BEGIN
   Info_Manag.P_Byte_First_Info := 20;
   Info_Manag.No_of_Infos := 30;
   Info_Manag.Len_Info := 24;
   Para_CMD[1].S_DB_No := 402;
   Para_CMD[1].S_Adress := 800;
   Para_CMD[1].D_Line := 1;
   Para_CMD[1].D_ASDU := 25860;
   Para_CMD[1].D_Info := 8;
   Para_CMD[1].Timeout := 10;
   Para_CMD[1].TI := 45;
   Para_CMD[1].Value := DWORD#16#0000_0005;
   Para_CMD[1].Termination_Type := 2;
   Para_CMD[2].S_DB_No := 402;
   Para_CMD[2].S_Adress := 816;
   Para_CMD[2].D_Line := 1;
   Para_CMD[2].D_ASDU := 25860;
   Para_CMD[2].D_Info := 9;
   Para_CMD[2].Timeout := 10;
   Para_CMD[2].TI := 45;
   Para_CMD[2].Value := DWORD#16#0000_0005;
   Para_CMD[2].Termination_Type := 2;
   Para_CMD[3].S_DB_No := 402;
   Para_CMD[3].S_Adress := 2016;
   Para_CMD[3].D_Line := 1;
   Para_CMD[3].D_ASDU := 26116;
   Para_CMD[3].D_Info := 8;
   Para_CMD[3].Timeout := 10;
   Para_CMD[3].TI := 45;
   Para_CMD[3].Value := DWORD#16#0000_0005;
   Para_CMD[3].Termination_Type := 2;
   Para_CMD[4].S_DB_No := 402;
   Para_CMD[4].S_Adress := 2032;
   Para_CMD[4].D_Line := 1;
   Para_CMD[4].D_ASDU := 26116;
   Para_CMD[4].D_Info := 9;
   Para_CMD[4].Timeout := 10;
   Para_CMD[4].TI := 45;
   Para_CMD[4].Value := DWORD#16#0000_0005;
   Para_CMD[4].Termination_Type := 2;
   Para_CMD[5].S_DB_No := 402;
   Para_CMD[5].S_Adress := 3232;
   Para_CMD[5].D_Line := 1;
   Para_CMD[5].D_ASDU := 26372;
   Para_CMD[5].D_Info := 8;
   Para_CMD[5].Timeout := 10;
   Para_CMD[5].TI := 45;
   Para_CMD[5].Value := DWORD#16#0000_0005;
   Para_CMD[5].Termination_Type := 2;
   Para_CMD[6].S_DB_No := 402;
   Para_CMD[6].S_Adress := 3248;
   Para_CMD[6].D_Line := 1;
   Para_CMD[6].D_ASDU := 26372;
   Para_CMD[6].D_Info := 9;
   Para_CMD[6].Timeout := 10;
   Para_CMD[6].TI := 45;
   Para_CMD[6].Value := DWORD#16#0000_0005;
   Para_CMD[6].Termination_Type := 2;
   Para_CMD[7].S_DB_No := 402;
   Para_CMD[7].S_Adress := 4448;
   Para_CMD[7].D_Line := 1;
   Para_CMD[7].D_ASDU := 26628;
   Para_CMD[7].D_Info := 8;
   Para_CMD[7].Timeout := 10;
   Para_CMD[7].TI := 45;
   Para_CMD[7].Value := DWORD#16#0000_0005;
   Para_CMD[7].Termination_Type := 2;
   Para_CMD[8].S_DB_No := 402;
   Para_CMD[8].S_Adress := 4464;
   Para_CMD[8].D_Line := 1;
   Para_CMD[8].D_ASDU := 26628;
   Para_CMD[8].D_Info := 9;
   Para_CMD[8].Timeout := 10;
   Para_CMD[8].TI := 45;
   Para_CMD[8].Value := DWORD#16#0000_0005;
   Para_CMD[8].Termination_Type := 2;
   Para_CMD[9].S_DB_No := 402;
   Para_CMD[9].S_Adress := 5664;
   Para_CMD[9].D_Line := 1;
   Para_CMD[9].D_ASDU := 26884;
   Para_CMD[9].D_Info := 8;
   Para_CMD[9].Timeout := 10;
   Para_CMD[9].TI := 45;
   Para_CMD[9].Value := DWORD#16#0000_0005;
   Para_CMD[9].Termination_Type := 2;
   Para_CMD[10].S_DB_No := 402;
   Para_CMD[10].S_Adress := 5680;
   Para_CMD[10].D_Line := 1;
   Para_CMD[10].D_ASDU := 26884;
   Para_CMD[10].D_Info := 9;
   Para_CMD[10].Timeout := 10;
   Para_CMD[10].TI := 45;
   Para_CMD[10].Value := DWORD#16#0000_0005;
   Para_CMD[10].Termination_Type := 2;
   Para_CMD[11].S_DB_No := 402;
   Para_CMD[11].S_Adress := 6880;
   Para_CMD[11].D_Line := 1;
   Para_CMD[11].D_ASDU := 27140;
   Para_CMD[11].D_Info := 8;
   Para_CMD[11].Timeout := 10;
   Para_CMD[11].TI := 45;
   Para_CMD[11].Value := DWORD#16#0000_0005;
   Para_CMD[11].Termination_Type := 2;
   Para_CMD[12].S_DB_No := 402;
   Para_CMD[12].S_Adress := 6896;
   Para_CMD[12].D_Line := 1;
   Para_CMD[12].D_ASDU := 27140;
   Para_CMD[12].D_Info := 9;
   Para_CMD[12].Timeout := 10;
   Para_CMD[12].TI := 45;
   Para_CMD[12].Value := DWORD#16#0000_0005;
   Para_CMD[12].Termination_Type := 2;
   Para_CMD[13].S_DB_No := 402;
   Para_CMD[13].S_Adress := 8096;
   Para_CMD[13].D_Line := 1;
   Para_CMD[13].D_ASDU := 27396;
   Para_CMD[13].D_Info := 8;
   Para_CMD[13].Timeout := 10;
   Para_CMD[13].TI := 45;
   Para_CMD[13].Value := DWORD#16#0000_0005;
   Para_CMD[13].Termination_Type := 2;
   Para_CMD[14].S_DB_No := 402;
   Para_CMD[14].S_Adress := 8112;
   Para_CMD[14].D_Line := 1;
   Para_CMD[14].D_ASDU := 27396;
   Para_CMD[14].D_Info := 9;
   Para_CMD[14].Timeout := 10;
   Para_CMD[14].TI := 45;
   Para_CMD[14].Value := DWORD#16#0000_0005;
   Para_CMD[14].Termination_Type := 2;
   Para_CMD[15].S_DB_No := 402;
   Para_CMD[15].S_Adress := 9312;
   Para_CMD[15].D_Line := 1;
   Para_CMD[15].D_ASDU := 27652;
   Para_CMD[15].D_Info := 8;
   Para_CMD[15].Timeout := 10;
   Para_CMD[15].TI := 45;
   Para_CMD[15].Value := DWORD#16#0000_0005;
   Para_CMD[15].Termination_Type := 2;
   Para_CMD[16].S_DB_No := 402;
   Para_CMD[16].S_Adress := 9328;
   Para_CMD[16].D_Line := 1;
   Para_CMD[16].D_ASDU := 27652;
   Para_CMD[16].D_Info := 9;
   Para_CMD[16].Timeout := 10;
   Para_CMD[16].TI := 45;
   Para_CMD[16].Value := DWORD#16#0000_0005;
   Para_CMD[16].Termination_Type := 2;
   Para_CMD[17].S_DB_No := 402;
   Para_CMD[17].S_Adress := 10528;
   Para_CMD[17].D_Line := 1;
   Para_CMD[17].D_ASDU := 28164;
   Para_CMD[17].D_Info := 8;
   Para_CMD[17].Timeout := 10;
   Para_CMD[17].TI := 45;
   Para_CMD[17].Value := DWORD#16#0000_0005;
   Para_CMD[17].Termination_Type := 2;
   Para_CMD[18].S_DB_No := 402;
   Para_CMD[18].S_Adress := 10544;
   Para_CMD[18].D_Line := 1;
   Para_CMD[18].D_ASDU := 28164;
   Para_CMD[18].D_Info := 9;
   Para_CMD[18].Timeout := 10;
   Para_CMD[18].TI := 45;
   Para_CMD[18].Value := DWORD#16#0000_0005;
   Para_CMD[18].Termination_Type := 2;
   Para_CMD[19].S_DB_No := 402;
   Para_CMD[19].S_Adress := 11744;
   Para_CMD[19].D_Line := 1;
   Para_CMD[19].D_ASDU := 28420;
   Para_CMD[19].D_Info := 8;
   Para_CMD[19].Timeout := 10;
   Para_CMD[19].TI := 45;
   Para_CMD[19].Value := DWORD#16#0000_0005;
   Para_CMD[19].Termination_Type := 2;
   Para_CMD[20].S_DB_No := 402;
   Para_CMD[20].S_Adress := 11760;
   Para_CMD[20].D_Line := 1;
   Para_CMD[20].D_ASDU := 28420;
   Para_CMD[20].D_Info := 9;
   Para_CMD[20].Timeout := 10;
   Para_CMD[20].TI := 45;
   Para_CMD[20].Value := DWORD#16#0000_0005;
   Para_CMD[20].Termination_Type := 2;
   Para_CMD[21].S_DB_No := 402;
   Para_CMD[21].S_Adress := 12960;
   Para_CMD[21].D_Line := 1;
   Para_CMD[21].D_ASDU := 28676;
   Para_CMD[21].D_Info := 8;
   Para_CMD[21].Timeout := 10;
   Para_CMD[21].TI := 45;
   Para_CMD[21].Value := DWORD#16#0000_0005;
   Para_CMD[21].Termination_Type := 2;
   Para_CMD[22].S_DB_No := 402;
   Para_CMD[22].S_Adress := 12976;
   Para_CMD[22].D_Line := 1;
   Para_CMD[22].D_ASDU := 28676;
   Para_CMD[22].D_Info := 9;
   Para_CMD[22].Timeout := 10;
   Para_CMD[22].TI := 45;
   Para_CMD[22].Value := DWORD#16#0000_0005;
   Para_CMD[22].Termination_Type := 2;
   Para_CMD[23].S_DB_No := 402;
   Para_CMD[23].S_Adress := 14176;
   Para_CMD[23].D_Line := 1;
   Para_CMD[23].D_ASDU := 28932;
   Para_CMD[23].D_Info := 8;
   Para_CMD[23].Timeout := 10;
   Para_CMD[23].TI := 45;
   Para_CMD[23].Value := DWORD#16#0000_0005;
   Para_CMD[23].Termination_Type := 2;
   Para_CMD[24].S_DB_No := 402;
   Para_CMD[24].S_Adress := 14192;
   Para_CMD[24].D_Line := 1;
   Para_CMD[24].D_ASDU := 28932;
   Para_CMD[24].D_Info := 9;
   Para_CMD[24].Timeout := 10;
   Para_CMD[24].TI := 45;
   Para_CMD[24].Value := DWORD#16#0000_0005;
   Para_CMD[24].Termination_Type := 2;
   Para_CMD[25].S_DB_No := 402;
   Para_CMD[25].S_Adress := 15392;
   Para_CMD[25].D_Line := 1;
   Para_CMD[25].D_ASDU := 29188;
   Para_CMD[25].D_Info := 8;
   Para_CMD[25].Timeout := 10;
   Para_CMD[25].TI := 45;
   Para_CMD[25].Value := DWORD#16#0000_0005;
   Para_CMD[25].Termination_Type := 2;
   Para_CMD[26].S_DB_No := 402;
   Para_CMD[26].S_Adress := 15408;
   Para_CMD[26].D_Line := 1;
   Para_CMD[26].D_ASDU := 29188;
   Para_CMD[26].D_Info := 9;
   Para_CMD[26].Timeout := 10;
   Para_CMD[26].TI := 45;
   Para_CMD[26].Value := DWORD#16#0000_0005;
   Para_CMD[26].Termination_Type := 2;
   Para_CMD[27].S_DB_No := 402;
   Para_CMD[27].S_Adress := 16608;
   Para_CMD[27].D_Line := 1;
   Para_CMD[27].D_ASDU := 30468;
   Para_CMD[27].D_Info := 8;
   Para_CMD[27].Timeout := 10;
   Para_CMD[27].TI := 45;
   Para_CMD[27].Value := DWORD#16#0000_0005;
   Para_CMD[27].Termination_Type := 2;
   Para_CMD[28].S_DB_No := 402;
   Para_CMD[28].S_Adress := 16624;
   Para_CMD[28].D_Line := 1;
   Para_CMD[28].D_ASDU := 30468;
   Para_CMD[28].D_Info := 9;
   Para_CMD[28].Timeout := 10;
   Para_CMD[28].TI := 45;
   Para_CMD[28].Value := DWORD#16#0000_0005;
   Para_CMD[28].Termination_Type := 2;
   Para_CMD[29].S_DB_No := 402;
   Para_CMD[29].S_Adress := 17824;
   Para_CMD[29].D_Line := 1;
   Para_CMD[29].D_ASDU := 5126;
   Para_CMD[29].D_Info := 8;
   Para_CMD[29].Timeout := 10;
   Para_CMD[29].TI := 45;
   Para_CMD[29].Value := DWORD#16#0000_0005;
   Para_CMD[29].Termination_Type := 2;
   Para_CMD[30].S_DB_No := 402;
   Para_CMD[30].S_Adress := 17840;
   Para_CMD[30].D_Line := 1;
   Para_CMD[30].D_ASDU := 5126;
   Para_CMD[30].D_Info := 9;
   Para_CMD[30].Timeout := 10;
   Para_CMD[30].TI := 45;
   Para_CMD[30].Value := DWORD#16#0000_0005;
   Para_CMD[30].Termination_Type := 2;

END_DATA_BLOCK

DATA_BLOCK "DB_IEC_Para_MAo_ME"
{ S7_Optimized_Access := 'FALSE' }
AUTHOR : SIE_GST
FAMILY : S7_IEC
NAME : P_NA_IM
VERSION : 1.6
   STRUCT
      DB_Manag { ExternalVisible := 'False'} : Struct
         Pos_of_DB { ExternalVisible := 'False'} : Byte;   // reserved for future - do not change !
         No_of_all_DBs { ExternalVisible := 'False'} : Byte;   // reserved for future - do not change !
         DB_No_Act { ExternalVisible := 'False'} : Word;   // reserved for future - do not change !
         DB_No_Prev { ExternalVisible := 'False'} : Word;   // reserved for future - do not change !
         DB_No_Next { ExternalVisible := 'False'} : Word;   // reserved for future - do not change !
         Reserved { ExternalVisible := 'False'} : Word;
      END_STRUCT;
      Info_Manag { ExternalVisible := 'False'} : Struct
         P_Byte_First_Info { ExternalVisible := 'False'} : Int;   // (Byte-) Position of first Para-Block - do not change !
         No_of_Infos { ExternalVisible := 'False'} : Int;   // 0:unspecified (DB is filled up to the end); otherwise size n of ARRAY [1..n]
         Len_Info { ExternalVisible := 'False'} : USInt;   // Difference in [byte] between two Para-Blocks - do not change !
         Len_Sort_Key { ExternalVisible := 'False'} : USInt;   // 0: without sorting; 1-8: Data sets are sorted ascending
         Re_internal_usage { ExternalVisible := 'False'} : DWord;
      END_STRUCT;
      Global { ExternalVisible := 'False'} : Struct
         Para_DB_Type { ExternalVisible := 'False'} : Word;   // Internal identifier for this Data Block - do not change
         Image_Type { ExternalVisible := 'False'} : Byte;   // 1: Measuered value 2 Bytes, 2: IEC,  3 IEC+Ext_State+Time
         Image_Len { ExternalVisible := 'False'} : Byte;   // 0: auto (standard); <> 0: fixed distance [Bit] of procesimages
         Subst_on_Error { ExternalVisible := 'False'} : Bool;   // Substitute values in case of connection errors ?
         Subst_Value { ExternalVisible := 'False'} : DWord;   // Substitute value (if activated).
         Internal_10 { ExternalVisible := 'False'} : Word;   // Internal use: Last found parablock - do not change !
         Internal_12 { ExternalVisible := 'False'} : Word;   // Internal use: Last processed info - do not change !
      END_STRUCT;
      Para { ExternalVisible := 'False'} : Array[1..60] of Struct
         S_Line { ExternalVisible := 'False'} : Int;   // Source (Quelle): No of Line (Nr der Linie) (1..x)-actually do not change from 1
         S_ASDU { ExternalVisible := 'False'} : UInt;   // Source (Quelle): Address of ASDU (ASDU-Adresse)
         S_Info { ExternalVisible := 'False'} : DInt;   // Source (Quelle): Address of Infoobject (IOA)
         D_DB_No { ExternalVisible := 'False'} : Int;   // Dest. (Ziel) No. of DataBlock, 0 -> PIQ (PAA)
         D_Address { ExternalVisible := 'False'} : DInt;   // Dest. (Ziel): Bitposition
         P_No_of_fol_Infos { ExternalVisible := 'False'} : Int;   // Parameter: Number of following sequ. Infoelements
      END_STRUCT;
   END_STRUCT;


BEGIN
   Info_Manag.P_Byte_First_Info := 34;
   Info_Manag.No_of_Infos := 60;
   Info_Manag.Len_Info := 16;
   Global.Para_DB_Type := WORD#16#0109;
   Global.Image_Type := BYTE#16#03;
   Para[1].S_Line := 1;
   Para[1].S_ASDU := 25860;
   Para[1].S_Info := 16;
   Para[1].D_DB_No := 402;
   Para[1].D_Address := 832;
   Para[2].S_Line := 1;
   Para[2].S_ASDU := 25860;
   Para[2].S_Info := 17;
   Para[2].D_DB_No := 402;
   Para[2].D_Address := 928;
   Para[3].S_Line := 1;
   Para[3].S_ASDU := 25860;
   Para[3].S_Info := 18;
   Para[3].D_DB_No := 402;
   Para[3].D_Address := 1024;
   Para[4].S_Line := 1;
   Para[4].S_ASDU := 25860;
   Para[4].S_Info := 19;
   Para[4].D_DB_No := 402;
   Para[4].D_Address := 1120;
   Para[5].S_Line := 1;
   Para[5].S_ASDU := 26116;
   Para[5].S_Info := 16;
   Para[5].D_DB_No := 402;
   Para[5].D_Address := 2048;
   Para[6].S_Line := 1;
   Para[6].S_ASDU := 26116;
   Para[6].S_Info := 17;
   Para[6].D_DB_No := 402;
   Para[6].D_Address := 2144;
   Para[7].S_Line := 1;
   Para[7].S_ASDU := 26116;
   Para[7].S_Info := 18;
   Para[7].D_DB_No := 402;
   Para[7].D_Address := 2240;
   Para[8].S_Line := 1;
   Para[8].S_ASDU := 26116;
   Para[8].S_Info := 19;
   Para[8].D_DB_No := 402;
   Para[8].D_Address := 2336;
   Para[9].S_Line := 1;
   Para[9].S_ASDU := 26372;
   Para[9].S_Info := 16;
   Para[9].D_DB_No := 402;
   Para[9].D_Address := 3264;
   Para[10].S_Line := 1;
   Para[10].S_ASDU := 26372;
   Para[10].S_Info := 17;
   Para[10].D_DB_No := 402;
   Para[10].D_Address := 3360;
   Para[11].S_Line := 1;
   Para[11].S_ASDU := 26372;
   Para[11].S_Info := 18;
   Para[11].D_DB_No := 402;
   Para[11].D_Address := 3456;
   Para[12].S_Line := 1;
   Para[12].S_ASDU := 26372;
   Para[12].S_Info := 19;
   Para[12].D_DB_No := 402;
   Para[12].D_Address := 3552;
   Para[13].S_Line := 1;
   Para[13].S_ASDU := 26628;
   Para[13].S_Info := 16;
   Para[13].D_DB_No := 402;
   Para[13].D_Address := 4480;
   Para[14].S_Line := 1;
   Para[14].S_ASDU := 26628;
   Para[14].S_Info := 17;
   Para[14].D_DB_No := 402;
   Para[14].D_Address := 4576;
   Para[15].S_Line := 1;
   Para[15].S_ASDU := 26628;
   Para[15].S_Info := 18;
   Para[15].D_DB_No := 402;
   Para[15].D_Address := 4672;
   Para[16].S_Line := 1;
   Para[16].S_ASDU := 26628;
   Para[16].S_Info := 19;
   Para[16].D_DB_No := 402;
   Para[16].D_Address := 4768;
   Para[17].S_Line := 1;
   Para[17].S_ASDU := 26884;
   Para[17].S_Info := 16;
   Para[17].D_DB_No := 402;
   Para[17].D_Address := 5696;
   Para[18].S_Line := 1;
   Para[18].S_ASDU := 26884;
   Para[18].S_Info := 17;
   Para[18].D_DB_No := 402;
   Para[18].D_Address := 5792;
   Para[19].S_Line := 1;
   Para[19].S_ASDU := 26884;
   Para[19].S_Info := 18;
   Para[19].D_DB_No := 402;
   Para[19].D_Address := 5888;
   Para[20].S_Line := 1;
   Para[20].S_ASDU := 26884;
   Para[20].S_Info := 19;
   Para[20].D_DB_No := 402;
   Para[20].D_Address := 5984;
   Para[21].S_Line := 1;
   Para[21].S_ASDU := 27140;
   Para[21].S_Info := 16;
   Para[21].D_DB_No := 402;
   Para[21].D_Address := 6912;
   Para[22].S_Line := 1;
   Para[22].S_ASDU := 27140;
   Para[22].S_Info := 17;
   Para[22].D_DB_No := 402;
   Para[22].D_Address := 7008;
   Para[23].S_Line := 1;
   Para[23].S_ASDU := 27140;
   Para[23].S_Info := 18;
   Para[23].D_DB_No := 402;
   Para[23].D_Address := 7104;
   Para[24].S_Line := 1;
   Para[24].S_ASDU := 27140;
   Para[24].S_Info := 19;
   Para[24].D_DB_No := 402;
   Para[24].D_Address := 7200;
   Para[25].S_Line := 1;
   Para[25].S_ASDU := 27396;
   Para[25].S_Info := 16;
   Para[25].D_DB_No := 402;
   Para[25].D_Address := 8128;
   Para[26].S_Line := 1;
   Para[26].S_ASDU := 27396;
   Para[26].S_Info := 17;
   Para[26].D_DB_No := 402;
   Para[26].D_Address := 8224;
   Para[27].S_Line := 1;
   Para[27].S_ASDU := 27396;
   Para[27].S_Info := 18;
   Para[27].D_DB_No := 402;
   Para[27].D_Address := 8320;
   Para[28].S_Line := 1;
   Para[28].S_ASDU := 27396;
   Para[28].S_Info := 19;
   Para[28].D_DB_No := 402;
   Para[28].D_Address := 8416;
   Para[29].S_Line := 1;
   Para[29].S_ASDU := 27652;
   Para[29].S_Info := 16;
   Para[29].D_DB_No := 402;
   Para[29].D_Address := 9344;
   Para[30].S_Line := 1;
   Para[30].S_ASDU := 27652;
   Para[30].S_Info := 17;
   Para[30].D_DB_No := 402;
   Para[30].D_Address := 9440;
   Para[31].S_Line := 1;
   Para[31].S_ASDU := 27652;
   Para[31].S_Info := 18;
   Para[31].D_DB_No := 402;
   Para[31].D_Address := 9536;
   Para[32].S_Line := 1;
   Para[32].S_ASDU := 27652;
   Para[32].S_Info := 19;
   Para[32].D_DB_No := 402;
   Para[32].D_Address := 9632;
   Para[33].S_Line := 1;
   Para[33].S_ASDU := 28164;
   Para[33].S_Info := 16;
   Para[33].D_DB_No := 402;
   Para[33].D_Address := 10560;
   Para[34].S_Line := 1;
   Para[34].S_ASDU := 28164;
   Para[34].S_Info := 17;
   Para[34].D_DB_No := 402;
   Para[34].D_Address := 10656;
   Para[35].S_Line := 1;
   Para[35].S_ASDU := 28164;
   Para[35].S_Info := 18;
   Para[35].D_DB_No := 402;
   Para[35].D_Address := 10752;
   Para[36].S_Line := 1;
   Para[36].S_ASDU := 28164;
   Para[36].S_Info := 19;
   Para[36].D_DB_No := 402;
   Para[36].D_Address := 10848;
   Para[37].S_Line := 1;
   Para[37].S_ASDU := 28420;
   Para[37].S_Info := 16;
   Para[37].D_DB_No := 402;
   Para[37].D_Address := 11776;
   Para[38].S_Line := 1;
   Para[38].S_ASDU := 28420;
   Para[38].S_Info := 17;
   Para[38].D_DB_No := 402;
   Para[38].D_Address := 11872;
   Para[39].S_Line := 1;
   Para[39].S_ASDU := 28420;
   Para[39].S_Info := 18;
   Para[39].D_DB_No := 402;
   Para[39].D_Address := 11968;
   Para[40].S_Line := 1;
   Para[40].S_ASDU := 28420;
   Para[40].S_Info := 19;
   Para[40].D_DB_No := 402;
   Para[40].D_Address := 12064;
   Para[41].S_Line := 1;
   Para[41].S_ASDU := 28676;
   Para[41].S_Info := 16;
   Para[41].D_DB_No := 402;
   Para[41].D_Address := 12992;
   Para[42].S_Line := 1;
   Para[42].S_ASDU := 28676;
   Para[42].S_Info := 17;
   Para[42].D_DB_No := 402;
   Para[42].D_Address := 13088;
   Para[43].S_Line := 1;
   Para[43].S_ASDU := 28676;
   Para[43].S_Info := 18;
   Para[43].D_DB_No := 402;
   Para[43].D_Address := 13184;
   Para[44].S_Line := 1;
   Para[44].S_ASDU := 28676;
   Para[44].S_Info := 19;
   Para[44].D_DB_No := 402;
   Para[44].D_Address := 13280;
   Para[45].S_Line := 1;
   Para[45].S_ASDU := 28932;
   Para[45].S_Info := 16;
   Para[45].D_DB_No := 402;
   Para[45].D_Address := 14208;
   Para[46].S_Line := 1;
   Para[46].S_ASDU := 28932;
   Para[46].S_Info := 17;
   Para[46].D_DB_No := 402;
   Para[46].D_Address := 14304;
   Para[47].S_Line := 1;
   Para[47].S_ASDU := 28932;
   Para[47].S_Info := 18;
   Para[47].D_DB_No := 402;
   Para[47].D_Address := 14400;
   Para[48].S_Line := 1;
   Para[48].S_ASDU := 28932;
   Para[48].S_Info := 19;
   Para[48].D_DB_No := 402;
   Para[48].D_Address := 14496;
   Para[49].S_Line := 1;
   Para[49].S_ASDU := 29188;
   Para[49].S_Info := 16;
   Para[49].D_DB_No := 402;
   Para[49].D_Address := 15424;
   Para[50].S_Line := 1;
   Para[50].S_ASDU := 29188;
   Para[50].S_Info := 17;
   Para[50].D_DB_No := 402;
   Para[50].D_Address := 15520;
   Para[51].S_Line := 1;
   Para[51].S_ASDU := 29188;
   Para[51].S_Info := 18;
   Para[51].D_DB_No := 402;
   Para[51].D_Address := 15616;
   Para[52].S_Line := 1;
   Para[52].S_ASDU := 29188;
   Para[52].S_Info := 19;
   Para[52].D_DB_No := 402;
   Para[52].D_Address := 15712;
   Para[53].S_Line := 1;
   Para[53].S_ASDU := 30468;
   Para[53].S_Info := 16;
   Para[53].D_DB_No := 402;
   Para[53].D_Address := 16640;
   Para[54].S_Line := 1;
   Para[54].S_ASDU := 30468;
   Para[54].S_Info := 17;
   Para[54].D_DB_No := 402;
   Para[54].D_Address := 16736;
   Para[55].S_Line := 1;
   Para[55].S_ASDU := 30468;
   Para[55].S_Info := 18;
   Para[55].D_DB_No := 402;
   Para[55].D_Address := 16832;
   Para[56].S_Line := 1;
   Para[56].S_ASDU := 30468;
   Para[56].S_Info := 19;
   Para[56].D_DB_No := 402;
   Para[56].D_Address := 16928;
   Para[57].S_Line := 1;
   Para[57].S_ASDU := 5126;
   Para[57].S_Info := 16;
   Para[57].D_DB_No := 402;
   Para[57].D_Address := 17856;
   Para[58].S_Line := 1;
   Para[58].S_ASDU := 5126;
   Para[58].S_Info := 17;
   Para[58].D_DB_No := 402;
   Para[58].D_Address := 17952;
   Para[59].S_Line := 1;
   Para[59].S_ASDU := 5126;
   Para[59].S_Info := 18;
   Para[59].D_DB_No := 402;
   Para[59].D_Address := 18048;
   Para[60].S_Line := 1;
   Para[60].S_ASDU := 5126;
   Para[60].S_Info := 19;
   Para[60].D_DB_No := 402;
   Para[60].D_Address := 18144;

END_DATA_BLOCK

